INTERFACE I_Deserializable EXTENDS __SYSTEM.IQueryInterface

METHOD TryDeserializeFrom : BOOL
VAR_INPUT
	Deserializer : I_Deserializer;
END_VAR
END_METHOD

END_INTERFACE

(* stored: Version 1.1.0.1, ProductVersion 3.1.4024.12
   Itf I_Deserializable: Id {9d227ebf-74e8-01e7-232e-08e38cfeb002}
   Method TryDeserializeFrom: Id {9e81621a-60b2-035b-0ed1-bc0b3d68fab1} *)
